FUNCTION_BLOCK detection
  (* Standard: 61499-2 *)
  (* Version 0,1, 2015-00-16, Th?o, PC_THEO *)
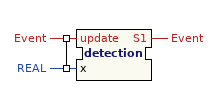
  EVENT_INPUT
    update WITH x;
  END_EVENT
  EVENT_OUTPUT
    S1;
  END_EVENT
  VAR_INPUT
    x : REAL;
  END_VAR
  VAR
    alpha : REAL;
  END_VAR
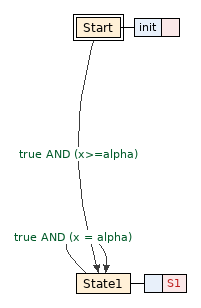
  EC_STATES
    Start : init;
    State1 : -> S1;
  END_STATES
  EC_TRANSITIONS
    Start TO State1 := true AND (x>=alpha);
    State1 TO State1 := true AND (x = alpha);
  END_TRANSITIONS
  ALGORITHM init IN C:
me->x=0;
me->alpha=3;
  END_ALGORITHM
END_FUNCTION_BLOCK
